{attribute 'qualified_only'}
{attribute 'strict'}
TYPE DUT_Permission :
(
    Hidden      := 0,
    ReadOnly    := 1,
    Write       := 2
);
END_TYPE

(* stored: Version 1.1.0.1, ProductVersion 3.1.4024.0
   DUT DUT_Permission: Id {d0d116a3-f331-42f4-9814-f49d528f871d} *)
